// TIA Portal V20 export
DATA_BLOCK "Mot"   // DB322
{ S7_Optimized_Access := 'TRUE' }
// stored: AutoNumber false, IsRetainMemResEnabled true, MemoryReserve 500, RetainMemoryReserve 500
   VAR RETAIN
      "8M1.B" : "TypeMotor";   // adjustment scanner
      "8M1.T" : "TypeMotor";   // adjustment top - normal drive
      "8M1.L" : "TypeMotor";   // adjustment left - normal drive
      "8M1.R" : "TypeMotor";   // adjustment right - normal drive
      "8U1.T" : "TypeMotor";   // adjustment top - linear drive
      "8U1.L" : "TypeMotor";   // adjustment left - linear drive
      "8U1.R" : "TypeMotor";   // adjustment right - linear drive
   END_VAR
BEGIN
   "8M1.B".description := WSTRING#'Motor Aufgabeförderer 1 - Zubringung';
   "8M1.T".description := WSTRING#'Motor Aufgabeförderer 2 - Zubringung';
   "8M1.L".description := WSTRING#'Motor Zerteiler - Zubringung';
   "8M1.R".description := WSTRING#'Motor Überbrückungsförderer - Zubringung';
   "8U1.T".description := WSTRING#'Motor Aufgabeförderer 2 - Zubringung';
   "8U1.L".description := WSTRING#'Motor Zerteiler - Zubringung';
   "8U1.R".description := WSTRING#'Motor Überbrückungsförderer - Zubringung';
END_DATA_BLOCK
